{attribute 'qualified_only'}
{attribute 'strict'}
TYPE eControlArchitectures :
(
	AggregatedLinear,
	CascadedWithElectricalCompensation,
	CascadedWithFullDecoupling,
	YET_TO_DEFINE
);
END_TYPE

(* stored: Version 1.1.0.1, ProductVersion 3.1.4024.12
   DUT eControlArchitectures: Id {24e8f4b4-b62c-47b7-9504-65ef2df06622} *)
